(* PLC project Tc2_Math.CEIL Demo, tc3-libraries-kb TwinCAT 3.1 *)
(* stored: creationDateTime 2026-05-10T10:00:00, modificationDateTime 2026-05-10T10:00:00 *)

PROGRAM P_Demo_CEIL
  VAR
    rResult : LREAL;  (* CEIL 的返回值 *)
    bRun : BOOL;  (* 触发一次调用 *)
  END_VAR

            // ============================================================
// Tc2_Math.CEIL 演示程序（FUNCTION）
// ============================================================
// 验证步骤：
//   1. 引用 Tc2_Math
//   2. 编译 + 登录
//   3. 强制 bRun := TRUE 一个周期
//   4. 在线监视 rResult 应为 3
// ============================================================

IF bRun THEN
    rResult := CEIL(2.8);
    bRun := FALSE;
END_IF;

          
END_PROGRAM
